(* IEC 61131-3 sources: Lasal/CPU_5344_V01/Class/Ram_CNC, 1 file *)

(* ---- Ram_CNC.st ---- *)
(*!
<Class
	Name               = "Ram_CNC"
	Revision           = "0.0"
	RealtimeTask       = "false"
	CyclicTask         = "false"
	BackgroundTask     = "false"
	Sigmatek           = "false"
	OSInterface        = "false"
	HighPriority       = "false"
	Automatic          = "false"
	UpdateMode         = "Prescan"
	SharedCommandTable = "true"
	Objectsize         = "(388,120)">
	<Channels>
		<Server Name="ActHomePos" Visualized="false" Initialize="false" WriteProtected="true" Retentive="false"/>
		<Server Name="ActMaxPos" Visualized="false" Initialize="false" WriteProtected="true" Retentive="false"/>
		<Server Name="ActMinPos" Visualized="false" Initialize="false" WriteProtected="true" Retentive="false"/>
		<Server Name="Afronding" Visualized="true" Initialize="false" WriteProtected="false" Retentive="SRam"/>
		<Server Name="Amax" Visualized="true" Initialize="false" WriteProtected="false" Retentive="SRam"/>
		<Server Name="DragLim" Visualized="true" Initialize="false" WriteProtected="false" Retentive="File"/>
		<Server Name="ExtUnits" Visualized="true" Initialize="false" WriteProtected="false" Retentive="File"/>
		<Server Name="HomePos" Visualized="true" Initialize="false" WriteProtected="false" Retentive="SRam"/>
		<Server Name="InPosBand" Visualized="true" Initialize="false" WriteProtected="false" Retentive="SRam"/>
		<Server Name="IntUnits" Visualized="true" Initialize="false" WriteProtected="false" Retentive="File"/>
		<Server Name="Kd" Visualized="true" Initialize="false" WriteProtected="false" Retentive="SRam"/>
		<Server Name="Ki" Visualized="true" Initialize="false" WriteProtected="false" Retentive="false"/>
		<Server Name="KISafe" Visualized="true" Initialize="false" WriteProtected="false" Retentive="SRam"/>
		<Server Name="Kv" Visualized="true" Initialize="false" WriteProtected="false" Retentive="SRam"/>
		<Server Name="lengteNeusstuk" Visualized="true" Initialize="false" WriteProtected="false" Retentive="SRam"/>
		<Server Name="MaxDecAs" Visualized="true" Initialize="false" WriteProtected="false" Retentive="SRam"/>
		<Server Name="MaxSignal" Visualized="true" Initialize="false" WriteProtected="false" Retentive="SRam"/>
		<Server Name="MaxSpeed" Visualized="true" Initialize="false" WriteProtected="false" Retentive="SRam"/>
		<Server Name="NeusstukActief" Visualized="true" Initialize="false" WriteProtected="false" Retentive="SRam"/>
		<Server Name="NullenAfrondingEnPosband" Visualized="true" Initialize="false" WriteProtected="true" Retentive="false"/>
		<Server Name="RefAcc" Visualized="true" Initialize="false" WriteProtected="false" Retentive="SRam"/>
		<Server Name="RefRichting" Visualized="true" Initialize="false" WriteProtected="false" Retentive="SRam"/>
		<Server Name="RefSpeed1" Visualized="true" Initialize="false" WriteProtected="false" Retentive="SRam"/>
		<Server Name="RefSpeed2" Visualized="true" Initialize="false" WriteProtected="false" Retentive="SRam"/>
		<Server Name="RemActief" Visualized="true" Initialize="false" WriteProtected="false" Retentive="SRam"/>
		<Server Name="Richting" Visualized="true" Initialize="false" WriteProtected="false" Retentive="SRam"/>
		<Server Name="SW_MaxPos" Visualized="true" Initialize="false" WriteProtected="false" Retentive="SRam"/>
		<Server Name="SW_MinPos" Visualized="true" Initialize="false" WriteProtected="false" Retentive="SRam"/>
		<Server Name="TijdRemLos" Visualized="true" Initialize="false" WriteProtected="false" Retentive="SRam"/>
		<Server Name="TijdRemVast" Visualized="true" Initialize="false" WriteProtected="false" Retentive="SRam"/>
		<Server Name="Vmax" Visualized="true" Initialize="false" WriteProtected="false" Retentive="SRam"/>
		<Server Name="Vu" Visualized="true" Initialize="false" WriteProtected="false" Retentive="SRam"/>
		<Server Name="XtraIfactor" Visualized="true" Initialize="false" WriteProtected="false" Retentive="SRam"/>
		<Server Name="XtraIWindow" Visualized="true" Initialize="false" WriteProtected="false" Retentive="SRam"/>
		<Client Name="AMaxWr" Required="true" Internal="false"/>
		<Client Name="cAmax" Required="false" Internal="false"/>
		<Client Name="cDragLim" Required="false" Internal="false"/>
		<Client Name="cExtUnits" Required="false" Internal="false"/>
		<Client Name="cHomePos" Required="false" Internal="false"/>
		<Client Name="cIntUnits" Required="false" Internal="false"/>
		<Client Name="cKv" Required="false" Internal="false"/>
		<Client Name="cMaxSignal" Required="false" Internal="false"/>
		<Client Name="cMaxSpeed" Required="false" Internal="false"/>
		<Client Name="cRefAcc" Required="false" Internal="false"/>
		<Client Name="cRefRichting" Required="true" Internal="false"/>
		<Client Name="cRefSpeed1" Required="false" Internal="false"/>
		<Client Name="cRefSpeed2" Required="false" Internal="false"/>
		<Client Name="cRichting" Required="false" Internal="false"/>
		<Client Name="cSw_MaxPos" Required="false" Internal="false"/>
		<Client Name="cVmax" Required="false" Internal="false"/>
		<Client Name="ExUnitsWr" Required="true" Internal="false"/>
		<Client Name="HomeOk" Required="true" Internal="false"/>
		<Client Name="IntUnitsWr" Required="true" Internal="false"/>
		<Client Name="MaxPosWr" Required="true" Internal="false"/>
		<Client Name="MinPosWr" Required="true" Internal="false"/>
		<Client Name="Resolutie" Required="true" Internal="false"/>
		<Client Name="VMaxWr" Required="true" Internal="false"/>
	</Channels>
	<Network Name="Ram_CNC">
		<!-- List of Components in this network -->
		<Components>
		</Components>
		<Comments>
		</Comments>
		<!-- List of Connections in this network -->
		<Connections>
		</Connections>
		<!-- Headerfiles -->
		<Options>
		</Options>
	</Network>
</Class>
*)
Ram_CNC : CLASS
  //Servers:
	ExtUnits 	: SvrChCmd_DINT;
	IntUnits 	: SvrChCmd_DINT;
	Vmax 	: SvrChCmd_DINT;
	Amax 	: SvrChCmd_DINT;
	MaxSpeed 	: SvrChCmd_DINT;
	Kv 	: SvrChCmd_DINT;
	Vu 	: SvrChCmd_DINT;
	Ki 	: SvrChCmd_DINT;
	Kd 	: SvrChCmd_DINT;
	DragLim 	: SvrChCmd_DINT;
	SW_MinPos 	: SvrCh_DINT;
	SW_MaxPos 	: SvrCh_DINT;
	HomePos 	: SvrCh_DINT;
	RefSpeed1 	: SvrCh_DINT;
	RefSpeed2 	: SvrCh_DINT;
	RefAcc 	: SvrCh_DINT;
	MaxSignal 	: SvrCh_DINT;
	Richting 	: SvrCh_DINT;
	RefRichting 	: SvrCh_DINT;
	KISafe 	: SvrCh_DINT;
	XtraIfactor 	: SvrCh_DINT;
	XtraIWindow 	: SvrCh_DINT;
	TijdRemVast 	: SvrCh_UDINT;
	TijdRemLos 	: SvrCh_UDINT;
	InPosBand 	: SvrCh_DINT;
	RemActief 	: SvrCh_DINT;
	Afronding 	: SvrCh_DINT;
	NullenAfrondingEnPosband 	: SvrCh_DINT;
	ActMinPos 	: SvrCh_DINT;
	ActMaxPos 	: SvrCh_DINT;
	ActHomePos 	: SvrCh_DINT;
	NeusstukActief 	: SvrCh_DINT;
	lengteNeusstuk 	: SvrCh_DINT;
	MaxDecAs 	: SvrCh_DINT;
  //Clients:
	cExtUnits 	: CltCh_DINT;
	cIntUnits 	: CltCh_DINT;
	cVmax 	: CltCh_DINT;
	cAmax 	: CltCh_DINT;
	cMaxSpeed 	: CltCh_DINT;
	cKv 	: CltCh_DINT;
	cDragLim 	: CltCh_DINT;
	cSw_MaxPos 	: CltCh_DINT;
	cHomePos 	: CltCh_DINT;
	cRefSpeed1 	: CltCh_DINT;
	cRefSpeed2 	: CltCh_DINT;
	cRefAcc 	: CltCh_DINT;
	cMaxSignal 	: CltCh_DINT;
	cRichting 	: CltCh_DINT;
	cRefRichting 	: CltCh_DINT;
	HomeOk 	: CltCh_DINT;
	ExUnitsWr 	: CltCh_DINT;
	IntUnitsWr 	: CltCh_DINT;
	VMaxWr 	: CltCh_DINT;
	AMaxWr 	: CltCh_DINT;
	Resolutie 	: CltCh_DINT;
	MinPosWr 	: CltCh_DINT;
	MaxPosWr 	: CltCh_DINT;
  //Variables:
		First 	: DINT;
  //Functions:

	FUNCTION VIRTUAL GLOBAL Init;

	FUNCTION Check;

	FUNCTION OerInit;

	FUNCTION ResetCNC;

	FUNCTION VIRTUAL GLOBAL ExtUnits::Write
		VAR_INPUT
			input (EAX) 	: DINT;
		END_VAR
		VAR_OUTPUT
			result (EAX) 	: DINT;
		END_VAR;

	FUNCTION VIRTUAL GLOBAL IntUnits::Write
		VAR_INPUT
			input (EAX) 	: DINT;
		END_VAR
		VAR_OUTPUT
			result (EAX) 	: DINT;
		END_VAR;

	FUNCTION VIRTUAL GLOBAL Vmax::Write
		VAR_INPUT
			input (EAX) 	: DINT;
		END_VAR
		VAR_OUTPUT
			result (EAX) 	: DINT;
		END_VAR;

	FUNCTION VIRTUAL GLOBAL Amax::Write
		VAR_INPUT
			input (EAX) 	: DINT;
		END_VAR
		VAR_OUTPUT
			result (EAX) 	: DINT;
		END_VAR;

	FUNCTION VIRTUAL GLOBAL SW_MinPos::Write
		VAR_INPUT
			input (EAX) 	: DINT;
		END_VAR
		VAR_OUTPUT
			result (EAX) 	: DINT;
		END_VAR;

	FUNCTION VIRTUAL GLOBAL SW_MaxPos::Write
		VAR_INPUT
			input (EAX) 	: DINT;
		END_VAR
		VAR_OUTPUT
			result (EAX) 	: DINT;
		END_VAR;

	FUNCTION VIRTUAL GLOBAL HomePos::Write
		VAR_INPUT
			input (EAX) 	: DINT;
		END_VAR
		VAR_OUTPUT
			result (EAX) 	: DINT;
		END_VAR;

	FUNCTION VIRTUAL GLOBAL MaxSignal::Write
		VAR_INPUT
			input (EAX) 	: DINT;
		END_VAR
		VAR_OUTPUT
			result (EAX) 	: DINT;
		END_VAR;

	FUNCTION VIRTUAL GLOBAL Richting::Write
		VAR_INPUT
			input (EAX) 	: DINT;
		END_VAR
		VAR_OUTPUT
			result (EAX) 	: DINT;
		END_VAR;

	FUNCTION VIRTUAL GLOBAL RefRichting::Write
		VAR_INPUT
			input (EAX) 	: DINT;
		END_VAR
		VAR_OUTPUT
			result (EAX) 	: DINT;
		END_VAR;

	FUNCTION VIRTUAL GLOBAL NeusstukActief::Write
		VAR_INPUT
			input (EAX) 	: DINT;
		END_VAR
		VAR_OUTPUT
			result (EAX) 	: DINT;
		END_VAR;

	FUNCTION VIRTUAL GLOBAL lengteNeusstuk::Write
		VAR_INPUT
			input (EAX) 	: DINT;
		END_VAR
		VAR_OUTPUT
			result (EAX) 	: DINT;
		END_VAR;
  //Tables:
	FUNCTION @STD
		VAR_OUTPUT
			ret_code	: CONFSTATES;
		END_VAR;
	FUNCTION GLOBAL TAB @CT_;
END_CLASS;

FUNCTION VIRTUAL GLOBAL Ram_CNC::Init

  If First= 0 Then
    OerInit();
    First := 1;
  End_If;

END_FUNCTION //VIRTUAL GLOBAL Ram_CNC::Init

FUNCTION Ram_CNC::OerInit

  if ExtUnits <> 0 then //wachten tot ext units niet meer nul zijn

    Resolutie := Resolutie.Read();
    if Resolutie = 1000 then
      NullenAfrondingEnPosband := 4;
    elsif Resolutie = 100 then
      NullenAfrondingEnPosband := 3;
    elsif Resolutie = 10 then
      NullenAfrondingEnPosband := 2;
    else
      NullenAfrondingEnPosband := 1;
    end_if;

    If ExtUnits= 0 Then
      cExtUnits 	  := cExtUnits.read();
      ExtUnits.Write(input:=cExtUnits);
    End_If;

    If IntUnits= 0 Then
      cIntUnits 	  := cIntUnits.read();
      IntUnits.Write(input:=cIntUnits);
    End_If;

    If Vmax= 0 Then
      cVmax 		    := cVmax.read();
      Vmax.Write(input:=cVmax);
    End_If;

    If Amax= 0 Then
      cAmax 		    := cAmax.read();
      Amax.Write(input:=cAmax);
    End_If;

    If MaxSpeed= 0 Then
      cMaxSpeed   	:= cMaxSpeed.read();
      MaxSpeed.Write(input:=cMaxSpeed);
    End_If;

    If Kv= 0 Then
      cKv 			    := cKv.read();
      Kv.Write(input:=cKv);
    End_If;

    If DragLim= 0 Then
      cDragLim 	    := cDragLim.read();
      DragLim.Write(input:=cDragLim);
    End_If;

    If SW_Maxpos= 0 Then
      cSW_Maxpos    := cSW_MaxPos.read();
      SW_Maxpos.Write(input:=cSw_MaxPos);
    End_If;

    If HomePos= 0 Then
      cHomePos      := cHomePos.read();
      HomePos.Write(input:=cHomePos);
    End_If;

    If RefSpeed1= 0 Then
      cRefSpeed1    := cRefSpeed1.read();
      RefSpeed1.Write(input:=cRefSpeed1);
    End_If;

    If RefSpeed2= 0 Then
      cRefSpeed2    := cRefSpeed2.read();
      RefSpeed2.Write(input:=cRefSpeed2);
    End_If;

    If RefAcc= 0 Then
      cRefAcc    	  := cRefAcc.read();
      RefAcc.Write(input:=cRefAcc);
    End_If;

    If MaxSignal= 0 Then
      cMaxSignal    := cMaxSignal.read();

      MaxSignal.Write(input:=cMaxSignal);

      //Default-Richting inlezen
      cRichting  := cRichting.read() And 2#1;
      Richting.Write(input:=cRichting And 2#1);

      //Default-Referentie Richting inlezen
      cRefRichting := cRefRichting.read() And 2#1;
      RefRichting.Write(input:=cRefRichting And 2#1);

    End_If;

    ExUnitsWr := ExtUnits;
    ExUnitsWr.Write(input:=ExUnitsWr);
    IntUnitsWr := IntUnits;
    IntUnitsWr.Write(input:=IntUnitsWr);
    VMaxWr :=Vmax;
    VMaxWr.Write(input:=VMaxWr);
    AMaxWr := Amax;
    AMaxWr.Write(input:=AMaxWr);
    MinPosWr := SW_MinPos - 10; //anders gaat de boel bij overshoot in error
    MinPosWr.Write(input:=MinPosWr);
    MaxPosWr := SW_MaxPos + 10; //anders gaat de boel bij overshoot in error
    MaxPosWr.Write(input:=MaxPosWr);
    Ki := KISafe;
  end_if;

  Check();
END_FUNCTION

FUNCTION Ram_CNC::Check

  If Richting = 0 then
    If IntUnits< 0 Then
      IntUnits.Write(input:=IntUnits*-1);
    End_If;

//    If MaxSignal< 0 Then
//      MaxSignal.Write(input:=MaxSignal* -1);
//    End_If;
//
  Else
    If IntUnits> 0 Then
      IntUnits.Write(input:=IntUnits* -1);
    End_If;
//
//    If MaxSignal> 0 Then
//      MaxSignal.Write(input:=MaxSignal* -1);
//    End_If;
//
//
  End_if;

  if NeusstukActief = 0 then
    ActHomePos := HomePos;
    ActMaxPos := SW_MaxPos;
    ActMinPos := SW_MinPos;
  else
    ActHomePos := HomePos - lengteNeusstuk;
    ActMaxPos := SW_MaxPos - lengteNeusstuk;
    ActMinPos := SW_MinPos - lengteNeusstuk;
  end_if;

END_FUNCTION

FUNCTION VIRTUAL GLOBAL Ram_CNC::ExtUnits::Write
	VAR_INPUT
		input (EAX) 	: DINT;
	END_VAR
	VAR_OUTPUT
		result (EAX) 	: DINT;
	END_VAR

  If Input<> 0 Then
    ExtUnits := input;
    result := ExtUnits;
    ExUnitsWr := ExtUnits;
    ExUnitsWr.Write(input:=ExUnitsWr);
    ResetCNC();
  Else
    Result  := Access_Denied;
  End_If;
END_FUNCTION //VIRTUAL GLOBAL Ram_CNC::ExtUnits::Write

FUNCTION VIRTUAL GLOBAL Ram_CNC::IntUnits::Write
VAR_INPUT
	input		: DINT;
END_VAR
VAR_OUTPUT
	result		: DINT;
END_VAR

  If Input> 0 Then
   If Richting= 0 Then
     IntUnits := input;
     result := IntUnits;
     ResetCNC();
    Else
      Result  := Access_Denied;
    End_If;
  ElsIf Input< 0 Then
    If Richting= 1 Then
      IntUnits := input;
      result := IntUnits;
      ResetCNC();
    Else
      Result  := Access_Denied;
    End_If;
  Else
    Result  := Access_Denied;
  End_If;

  IntUnitsWr := IntUnits;
  IntUnitsWr.Write(input:=IntUnitsWr);

END_FUNCTION //VIRTUAL GLOBAL Ram_CNC::IntUnits::Write

FUNCTION VIRTUAL GLOBAL Ram_CNC::Vmax::Write
VAR_INPUT
	input		: DINT;
END_VAR
VAR_OUTPUT
	result		: DINT;
END_VAR

	Vmax := input;
  VMaxWr := Vmax;
  VMaxWr.Write(input:=VMaxWr);
 	result := Vmax;

END_FUNCTION //VIRTUAL GLOBAL Ram_CNC::Vmax::Write

FUNCTION VIRTUAL GLOBAL Ram_CNC::Amax::Write
VAR_INPUT
	input		: DINT;
END_VAR
VAR_OUTPUT
	result		: DINT;
END_VAR

	Amax := input;
  AMaxWr := Amax;
  AMaxWr.Write(input:=AMaxWr);
 	result := Amax;

END_FUNCTION //VIRTUAL GLOBAL Ram_CNC::Amax::Write

 //VIRTUAL GLOBAL Ram_CNC::MaxSpeed::Write

 //VIRTUAL GLOBAL Ram_CNC::Kv::Write

 //VIRTUAL GLOBAL Ram_CNC::Vu::Write

 //VIRTUAL GLOBAL Ram_CNC::Ki::Write

 //VIRTUAL GLOBAL Ram_CNC::Kd::Write

 //VIRTUAL GLOBAL Ram_CNC::DragLim::Write

FUNCTION VIRTUAL GLOBAL Ram_CNC::SW_MinPos::Write
VAR_INPUT
	input		: DINT;
END_VAR
VAR_OUTPUT
	result		: DINT;
END_VAR

	SW_MinPos := input;
  MinPosWr := SW_MinPos - 10; //anders gaat de boel bij overshoot in error
  MinPosWr.Write(input:=MinPosWr);
 	result := SW_MinPos;
  ResetCNC();
  Check();

END_FUNCTION //VIRTUAL GLOBAL Ram_CNC::SW_MinPos::Write

FUNCTION VIRTUAL GLOBAL Ram_CNC::SW_MaxPos::Write
VAR_INPUT
	input		: DINT;
END_VAR
VAR_OUTPUT
	result		: DINT;
END_VAR

	SW_MaxPos := input;
  MaxPosWr := SW_MaxPos +10; //anders gaat de boel bij overshoot in error
  MaxPosWr.Write(input:=MaxPosWr);
 	result := SW_MaxPos;
  ResetCNC();
  Check();
END_FUNCTION //VIRTUAL GLOBAL Ram_CNC::SW_MaxPos::Write

 //VIRTUAL GLOBAL Ram_CNC::HomePos::Write

 //VIRTUAL GLOBAL Ram_CNC::RefSpeed1::Write

 //VIRTUAL GLOBAL Ram_CNC::RefSpeed2::Write

 //VIRTUAL GLOBAL Ram_CNC::RefAcc::Write

FUNCTION VIRTUAL GLOBAL Ram_CNC::MaxSignal::Write
	VAR_INPUT
		input (EAX) 	: DINT;
	END_VAR
	VAR_OUTPUT
		result (EAX) 	: DINT;
	END_VAR

//  If Input   > 0
//   & Richting= 0 Then
    MaxSignal := input;
    result := MaxSignal;
    ResetCNC();
//  ElsIf Input   < 0
//      & Richting= 1 Then
//    MaxSignal := input;
//    result := MaxSignal;
//    ResetCNC();
//  Else
//    Result  := Access_Denied;
//  End_If;
END_FUNCTION

FUNCTION VIRTUAL GLOBAL Ram_CNC::Richting::Write
VAR_INPUT
	input		: DINT;
END_VAR
VAR_OUTPUT
	result		: DINT;
END_VAR

	Richting := input And 2#1;
  Check();
  ResetCNC();
 	result := Richting;
END_FUNCTION //VIRTUAL GLOBAL Ram_CNC::Richting::Write

FUNCTION VIRTUAL GLOBAL Ram_CNC::RefRichting::Write
	VAR_INPUT
		input (EAX) 	: DINT;
	END_VAR
	VAR_OUTPUT
		result (EAX) 	: DINT;
	END_VAR

	RefRichting := input And 2#1;
 	result := RefRichting;
END_FUNCTION

FUNCTION Ram_CNC::ResetCNC

  HomeOk:=0;
  HomeOk.Write (HomeOk);

END_FUNCTION

FUNCTION VIRTUAL GLOBAL Ram_CNC::NeusstukActief::Write
	VAR_INPUT
		input (EAX) 	: DINT;
	END_VAR
	VAR_OUTPUT
		result (EAX) 	: DINT;
	END_VAR

  if input <> NeusstukActief then
	  NeusstukActief := input;
    Check();
    HomeOk.Write(input:=0);
  end_if;
	result := NeusstukActief;

END_FUNCTION

FUNCTION VIRTUAL GLOBAL Ram_CNC::lengteNeusstuk::Write
	VAR_INPUT
		input (EAX) 	: DINT;
	END_VAR
	VAR_OUTPUT
		result (EAX) 	: DINT;
	END_VAR

  if input <> lengteNeusstuk then

	  lengteNeusstuk := input;

    if NeusstukActief = 1 then
      Check();
      HomeOk.Write(input:=0);
    end_if;
  end_if;

	result := lengteNeusstuk;

END_FUNCTION

FUNCTION VIRTUAL GLOBAL Ram_CNC::HomePos::Write
	VAR_INPUT
		input (EAX) 	: DINT;
	END_VAR
	VAR_OUTPUT
		result (EAX) 	: DINT;
	END_VAR

	HomePos := input;
	result := HomePos;
  Check();

END_FUNCTION
